FUNCTION_BLOCK FB_Motor
VAR_INPUT
	mxReset							: BOOL;
	mxEmergency						: BOOL;
	mxAutoMode						: BOOL;
	mxDisableManualAutoTrigger		: BOOL := FALSE; // If this bit is enabled, the outputs status is not changed when change from/to automode happens
END_VAR
VAR_OUTPUT
(*Errors*)
	Errors							: ST_MotorErrors;
	mxErrorInit						: BOOL;		(* Error, stop immediately. Initialisation neccesary *)
	mxErrorStopinPos				: BOOL;		(* Error, stop in position. Only reset neccesary *)

(* State vars *)
	mxCycleBusy						: BOOL;
	mxInitBusy						: BOOL;
	
(* Vars *)
	mxInitialized					: BOOL;
	IsRunning						: BOOL;
	
END_VAR
VAR
	ixThermal						AT %I* : BOOL;
	ixRunning						AT %I* : BOOL;
	ixMaintenance					AT %I* : BOOL;
	Q								AT %Q* : BOOL;
	
	Hmi_On							: BOOL;
	RT_AutoMode						: R_TRIG;
	SR_ErrorThermal					: SR;
	SR_ErrorMaintenance				: SR;
	Ixtest: BOOL;
END_VAR

Error();

(* Reset hmi when switched to automode*)
RT_AutoMode(CLK:= mxAutoMode);

// if manual mode becomes active, the manualmode (hmi) is over written by its current state.
// this ensures that the motor keeps running when it was running and is switched to manual. 
IF RT_AutoMode.Q AND NOT mxDisableManualAutoTrigger THEN Hmi_On:= Q; END_IF	

(* Manual control *)
//IF NOT mxAutoMode THEN Q:= Hmi_On; END_IF

// Is running becomes high when signal becomes low.
IsRunning:= NOT ixRunning;

ACTION Error:
SR_ErrorThermal(SET1:= NOT ixThermal, RESET:= mxReset, Q1=> Errors.Thermal);
SR_ErrorMaintenance(SET1:= NOT ixMaintenance, RESET:= mxReset, Q1=> Errors.Maintenance);

(******************************************************************************************************)
mxErrorStopinPos:= FALSE;
mxErrorInit:= Errors.Thermal OR Errors.Maintenance;
END_ACTION

METHOD M_Init

Q:= FALSE;
END_METHOD

METHOD M_Start : BOOL
VAR_INPUT
END_VAR
Q:=TRUE;

(* Return Value *)
M_Start:= Q;
END_METHOD

METHOD M_Stop : BOOL
VAR_INPUT
END_VAR
Q:= FALSE;

(* Return Value *)
M_Stop:= NOT Q;
END_METHOD

END_FUNCTION_BLOCK

(* stored: Version 1.1.0.1, ProductVersion 3.1.4020.12
   POU FB_Motor: Id {dccc3e6f-a5bb-4f57-896d-021bb5c2e147}, SpecialFunc None
   Action Error: Id {4eac1137-ff38-460e-ba84-b81dd3446ebe}
   Method M_Init: Id {fde6f22f-b713-42ec-ae0a-377d2254630d}
   Method M_Start: Id {79110aac-879f-40af-9cd3-84457a8c1fff}
   Method M_Stop: Id {4a9aca0a-dd7a-4bb5-b3e9-ef23a97c2074} *)
